// Mitsubishi GX Works2 project: Assembler_Work   PLC: FX3U/FX3UC

PROGRAM MAIN
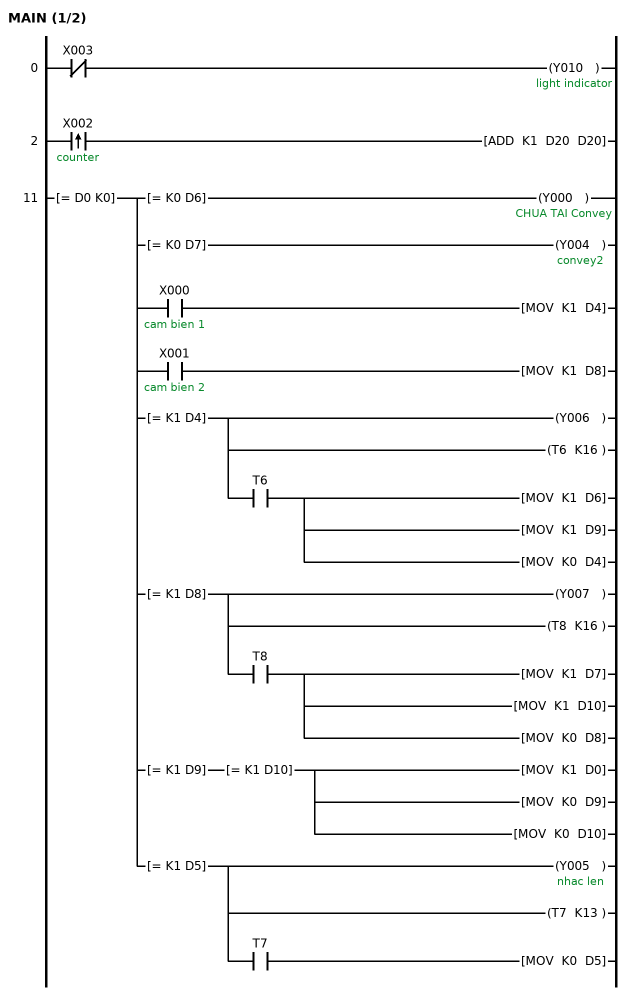
0     LDI     X003
      OUT     Y010  ; light indicator
2     LDP     X002  ; counter
      ADD     K1 D20 D20
11    LD=     D0 K0
      MPS
      AND=    K0 D6
      OUT     Y000  ; CHUA TAI Convey
      MRD
      AND=    K0 D7
      OUT     Y004  ; convey2
      MRD
      AND     X000  ; cam bien 1
      MOV     K1 D4
      MRD
      AND     X001  ; cam bien 2
      MOV     K1 D8
      MRD
      AND=    K1 D4
      OUT     Y006
      OUT     T6 K16
      AND     T6
      MOV     K1 D6
      MOV     K1 D9
      MOV     K0 D4
      MRD
      AND=    K1 D8
      OUT     Y007
      OUT     T8 K16
      AND     T8
      MOV     K1 D7
      MOV     K1 D10
      MOV     K0 D8
      MRD
      AND=    K1 D9
      AND=    K1 D10
      MOV     K1 D0
      MOV     K0 D9
      MOV     K0 D10
      MPP
      AND=    K1 D5
      OUT     Y005  ; nhac len
      OUT     T7 K13
      AND     T7
      MOV     K0 D5
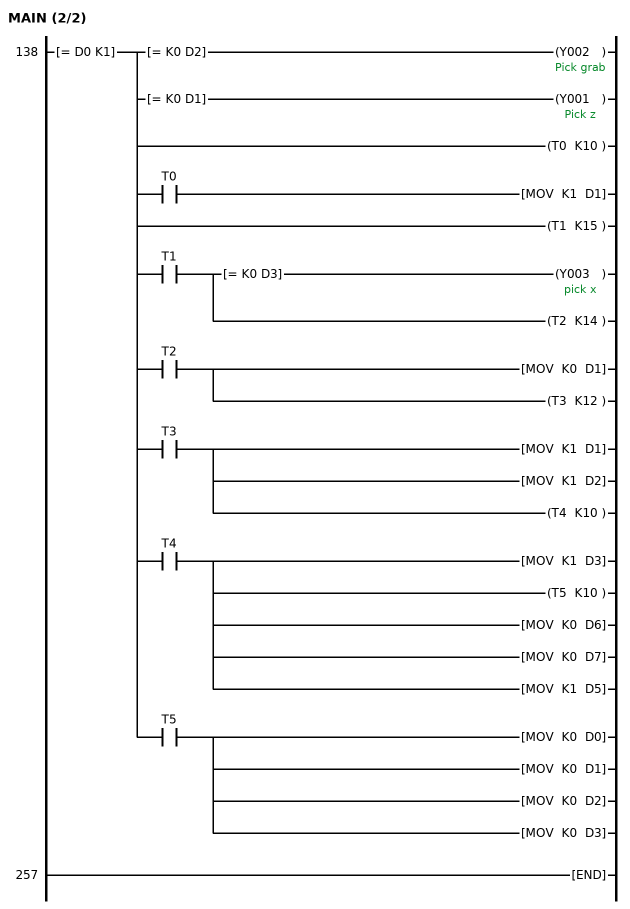
138   LD=     D0 K1
      MPS
      AND=    K0 D2
      OUT     Y002  ; Pick grab
      MRD
      AND=    K0 D1
      OUT     Y001  ; Pick z
      MPP
      OUT     T0 K10
      MPS
      AND     T0
      MOV     K1 D1
      MPP
      OUT     T1 K15
      MPS
      AND     T1
      MPS
      AND=    K0 D3
      OUT     Y003  ; pick x
      MPP
      OUT     T2 K14
      MRD
      AND     T2
      MOV     K0 D1
      OUT     T3 K12
      MRD
      AND     T3
      MOV     K1 D1
      MOV     K1 D2
      OUT     T4 K10
      MRD
      AND     T4
      MOV     K1 D3
      OUT     T5 K10
      MOV     K0 D6
      MOV     K0 D7
      MOV     K1 D5
      MPP
      AND     T5
      MOV     K0 D0
      MOV     K0 D1
      MOV     K0 D2
      MOV     K0 D3
257   END
END_PROGRAM

// device comments not shown above
X005  ; diffuse 4
X007  ; diffuse 4
Y011  ; auto curv1
Y012  ; spin+
Y013  ; pusher
Y014  ; auto 2m
Y015  ; 2m auto
Y016  ; pick 3z
Y017  ; pick 3 grab
Y020  ; pick 3 rotate cw
Y021  ; pick 3 rotate ccw
Y022  ; roller auto1
Y023  ; roller auto 2
Y024  ; roller auto 3
Y025  ; roller auto 4
Y026  ; roller auto 5
Y027  ; roller auto 6
D30  ; digital display
